FUNCTION_BLOCK FB_LamparaMemorizada_LD
// La lampara se enciende al accionar el pulsador de conexion
// La lampara se apaga al accionar el pulsador de desconexion
VAR
    Lampara              AT %Q*  : BOOL;
    PulsadorConexion     AT %I*  : BOOL;
    PulsadorDesconexion  AT %I*  : BOOL;
END_VAR

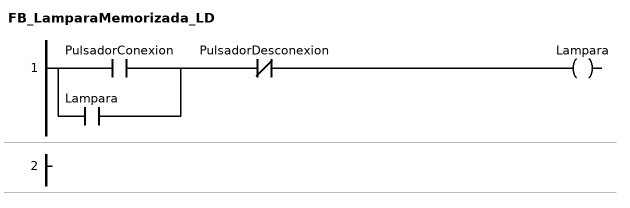
// NETWORK 1
Lampara := (PulsadorConexion OR Lampara) AND NOT PulsadorDesconexion;

// NETWORK 2

END_FUNCTION_BLOCK

(* stored: Version 1.1.0.1, ProductVersion 3.1.4024.15
   POU FB_LamparaMemorizada_LD: Id {3b068606-e4ed-4fff-8c23-37f5b0fb622b}, SpecialFunc None *)
